FUNCTION_BLOCK FB_FMS205_F1Producir_SFC EXTENDS FB_ControllerBase_SFC
VAR_IN_OUT
	Alime			: FB_Alimentador;
	Carga		 	: FB_PickAndPlace;
	Medid			: FB_MedidorTapa;
	Induc		 	: FB_CaptadorInductivo;
	Fotoe			: FB_DetectorFotoelectrico;
	Evacu		 	: FB_Evacuador;
	Desca			: FB_PickAndPlace;
	Plato			: FB_PlatoDivisor;
	Cinta			: FB_Cinta;
END_VAR

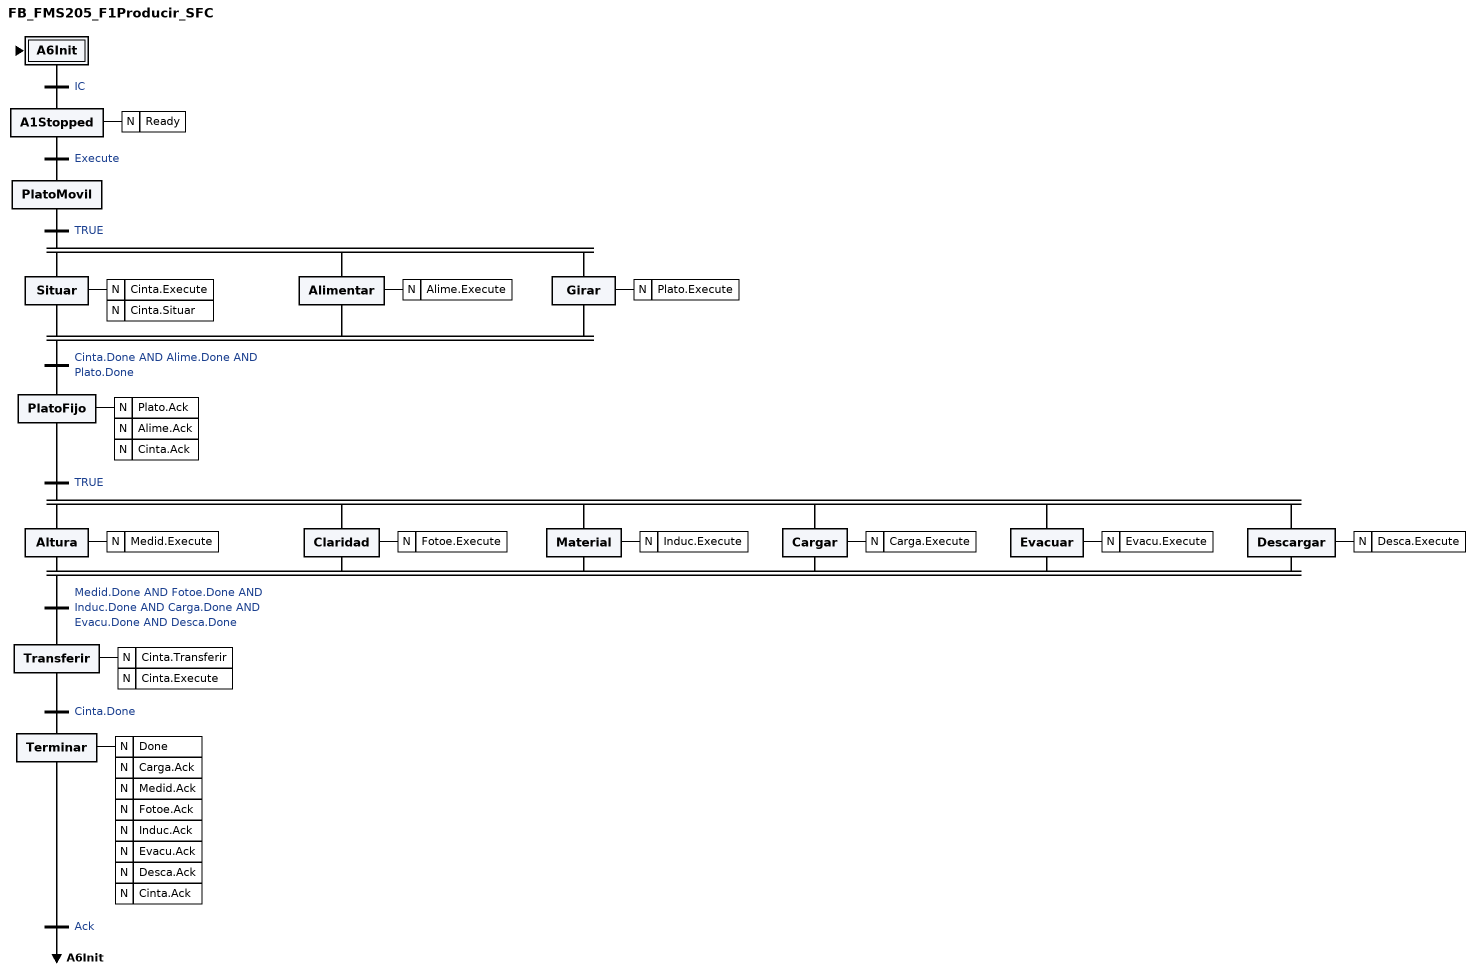
INITIAL_STEP A6Init:
END_STEP
TRANSITION FROM A6Init TO A1Stopped
    := IC;
END_TRANSITION
STEP A1Stopped:
    Ready(N);
END_STEP
TRANSITION FROM A1Stopped TO PlatoMovil
    := Execute;
END_TRANSITION
STEP PlatoMovil:
END_STEP
TRANSITION FROM PlatoMovil TO (Situar, Alimentar, Girar)
    := TRUE;
END_TRANSITION
STEP Situar:
    Cinta.Execute(N);
    Cinta.Situar(N);
END_STEP
STEP Alimentar:
    Alime.Execute(N);
END_STEP
STEP Girar:
    Plato.Execute(N);
END_STEP
TRANSITION FROM (Situar, Alimentar, Girar) TO PlatoFijo
    := Cinta.Done AND Alime.Done AND Plato.Done;
END_TRANSITION
STEP PlatoFijo:
    Plato.Ack(N);
    Alime.Ack(N);
    Cinta.Ack(N);
END_STEP
TRANSITION FROM PlatoFijo TO (Altura, Claridad, Material, Cargar, Evacuar, Descargar)
    := TRUE;
END_TRANSITION
STEP Altura:
    Medid.Execute(N);
END_STEP
STEP Claridad:
    Fotoe.Execute(N);
END_STEP
STEP Material:
    Induc.Execute(N);
END_STEP
STEP Cargar:
    Carga.Execute(N);
END_STEP
STEP Evacuar:
    Evacu.Execute(N);
END_STEP
STEP Descargar:
    Desca.Execute(N);
END_STEP
TRANSITION FROM (Altura, Claridad, Material, Cargar, Evacuar, Descargar) TO Transferir
    := Medid.Done AND Fotoe.Done AND Induc.Done AND Carga.Done AND Evacu.Done AND Desca.Done;
END_TRANSITION
STEP Transferir:
    Cinta.Transferir(N);
    Cinta.Execute(N);
END_STEP
TRANSITION FROM Transferir TO Terminar
    := Cinta.Done;
END_TRANSITION
STEP Terminar:
    Done(N);
    Carga.Ack(N);
    Medid.Ack(N);
    Fotoe.Ack(N);
    Induc.Ack(N);
    Evacu.Ack(N);
    Desca.Ack(N);
    Cinta.Ack(N);
END_STEP
TRANSITION FROM Terminar TO A6Init
    := Ack;
END_TRANSITION

END_FUNCTION_BLOCK

(* stored: Version 1.1.0.1, ProductVersion 3.1.4024.6
   POU FB_FMS205_F1Producir_SFC: Id {3765931f-4c2c-4236-9e0f-0066856caec5}, SpecialFunc None *)
